(* PLC project CoDeSys External Library Template, WAGO e!COCKPIT e!COCKPIT, author 3S - Smart Software Solutions GmbH *)
(* stored: creationDateTime 2019-10-29T12:37:19.3519458, version 3.5.5.30, modificationDateTime 2019-10-29T12:36:39.3744516, organization 3S - Smart Software Solutions GmbH *)
(* Library project template with all possible element types, docu and a sample project structure *)

(* values of enumPPPSFriskoATTOM1SError: BrakKomunikacji: brak komunikacji z węzłem; AlarmCzujnikaZewnetrznego: alarm braku zmiany wartości czujnika temp. zewnetrznj; AlarmCzujnikaZasilaniaObwoduCO: alarm braku zmiany wartości czujnika temp. zasilana obwod c. o.; BrakOsiagnieciaTemperaturyCO: alarm braku osiągnięcia temp. zadanej obwodu c. o.; BladIloscPomiarowTemperatury: alarm zbyt małej ilości pomiarów dokonanych w ciągu dnia do obliczenia średniej *)

(* Autor: Artur Wyszomirski, 2019-02-05-AWy Prawa majątkowe: Solwena Sp. z o.o., Aktualizacje: 2019-02-19-AWy: dodanie alarmów czujnika zew., zasilania c.o., braku osiągnięcia temperatury zadanej Opis: enum służy do obsługi alarmów w fb węzła Frisko ATTOM1S na budynkach PPP Sopot (ENGIE) *)
{attribute 'qualified_only'}
{attribute 'strict'}
TYPE enumPPPSFriskoATTOM1SError : (BrakKomunikacji := 1, AlarmCzujnikaZewnetrznego := 2, AlarmCzujnikaZasilaniaObwoduCO := 3, BrakOsiagnieciaTemperaturyCO := 4, BladIloscPomiarowTemperatury := 5);
END_TYPE
